//{attribute 'qualified_only'}
//{attribute 'strict'}
TYPE E_CounterReaction :
(
	eCounterReaction_None := 0,
	eCounterReaction_Info,
	eCounterReaction_Warning,
	eCounterReaction_Error,
	eCounterReaction_SerialFault_Warning,
	eCounterReaction_SerialFault_Error,
	
	eCounterReaction_Max
);
END_TYPE

(* stored: Version 1.1.0.1
   EnumerationTextList E_CounterReaction: Id {6a01f343-a4b3-41f2-9249-59e6192c2e25} *)
